// TIA Portal V18 export
DATA_BLOCK "DiagnosticTags"   // DB9
{ S7_Optimized_Access := 'TRUE' }
VERSION : 0.1
// stored: AutoNumber true, DBAccessibleFromOPCUA true, DBAccessibleFromWebserver true
   VAR
      "S1.CABINET000.STATE" : UDInt;
      "S1.CABINET001.STATE" : UDInt;
      "S1.CABINET002.STATE" : UDInt;
      "S1.CABINET003.STATE" : UDInt;
      "S1.CABINET015.STATE" : UDInt;
      "S1.CABINET014.STATE" : UDInt;
      "S1.CABINET012.STATE" : UDInt;
      "S1.CABINET013.STATE" : UDInt;
      "S1.CABINET004.STATE" : UDInt;
      "S1.CABINET011.STATE" : UDInt;
      "S1.CABINET010.STATE" : UDInt;
      "S1.CABINET009.STATE" : UDInt;
      "S1.CABINET005.STATE" : UDInt;
      "S1.CABINET006.STATE" : UDInt;
      "S1.CABINET007.STATE" : UDInt;
      "S1.CABINET008.STATE" : UDInt;
      "S1.CABINET000.ALARM1" : UDInt;
      "S1.CABINET001.ALARM1" : UDInt;
      "S1.CABINET002.ALARM1" : UDInt;
      "S1.CABINET003.ALARM1" : UDInt;
      "S1.CABINET015.ALARM1" : UDInt;
      "S1.CABINET014.ALARM1" : UDInt;
      "S1.CABINET012.ALARM1" : UDInt;
      "S1.CABINET013.ALARM1" : UDInt;
      "S1.CABINET004.ALARM1" : UDInt;
      "S1.CABINET011.ALARM1" : UDInt;
      "S1.CABINET010.ALARM1" : UDInt;
      "S1.CABINET009.ALARM1" : UDInt;
      "S1.CABINET005.ALARM1" : UDInt;
      "S1.CABINET006.ALARM1" : UDInt;
      "S1.CABINET007.ALARM1" : UDInt;
      "S1.CABINET008.ALARM1" : UDInt;
      "S1.CABINET000.ALARM2" : UDInt;
      "S1.CABINET001.ALARM2" : UDInt;
      "S1.CABINET002.ALARM2" : UDInt;
      "S1.CABINET003.ALARM2" : UDInt;
      "S1.CABINET015.ALARM2" : UDInt;
      "S1.CABINET014.ALARM2" : UDInt;
      "S1.CABINET012.ALARM2" : UDInt;
      "S1.CABINET013.ALARM2" : UDInt;
      "S1.CABINET004.ALARM2" : UDInt;
      "S1.CABINET011.ALARM2" : UDInt;
      "S1.CABINET010.ALARM2" : UDInt;
      "S1.CABINET009.ALARM2" : UDInt;
      "S1.CABINET005.ALARM2" : UDInt;
      "S1.CABINET006.ALARM2" : UDInt;
      "S1.CABINET007.ALARM2" : UDInt;
      "S1.CABINET008.ALARM2" : UDInt;
      "S1.CABINET000.WARNING1" : UDInt;
      "S1.CABINET001.WARNING1" : UDInt;
      "S1.CABINET002.WARNING1" : UDInt;
      "S1.CABINET003.WARNING1" : UDInt;
      "S1.CABINET015.WARNING1" : UDInt;
      "S1.CABINET014.WARNING1" : UDInt;
      "S1.CABINET012.WARNING1" : UDInt;
      "S1.CABINET013.WARNING1" : UDInt;
      "S1.CABINET004.WARNING1" : UDInt;
      "S1.CABINET011.WARNING1" : UDInt;
      "S1.CABINET010.WARNING1" : UDInt;
      "S1.CABINET009.WARNING1" : UDInt;
      "S1.CABINET005.WARNING1" : UDInt;
      "S1.CABINET006.WARNING1" : UDInt;
      "S1.CABINET007.WARNING1" : UDInt;
      "S1.CABINET008.WARNING1" : UDInt;
      "S1.CABINET000.WARNING2" : UDInt;
      "S1.CABINET001.WARNING2" : UDInt;
      "S1.CABINET002.WARNING2" : UDInt;
      "S1.CABINET003.WARNING2" : UDInt;
      "S1.CABINET015.WARNING2" : UDInt;
      "S1.CABINET014.WARNING2" : UDInt;
      "S1.CABINET012.WARNING2" : UDInt;
      "S1.CABINET013.WARNING2" : UDInt;
      "S1.CABINET004.WARNING2" : UDInt;
      "S1.CABINET011.WARNING2" : UDInt;
      "S1.CABINET010.WARNING2" : UDInt;
      "S1.CABINET009.WARNING2" : UDInt;
      "S1.CABINET005.WARNING2" : UDInt;
      "S1.CABINET006.WARNING2" : UDInt;
      "S1.CABINET007.WARNING2" : UDInt;
      "S1.CABINET008.WARNING2" : UDInt;
   END_VAR
BEGIN
END_DATA_BLOCK
